// TIA Portal project "Andon L1" (V14)

(* hardware
DEVICE "S7-1200 station_1"  S7-1200 Station
   slot 0: "Rack_0"  S7-1200 Rack  Rack  V1.0
   slot 1: "PLC_1"  CPU 1215C DC/DC/Rly  6ES7 215-1HG40-0XB0  V4.1
*)

// ===== PLC "PLC_1"  CPU 1215C DC/DC/Rly =====

VAR_GLOBAL   // PLC tag table "Default tag table"
   "inverterAssy" AT %I0.0 : Bool;
   "resetTimer" AT %I0.1 : Bool;
   "Tag_3" AT %I0.2 : Bool;
   "System_Byte" AT %MB1 : Byte;
   "FirstScan" AT %M1.0 : Bool;
   "DiagStatusUpdate" AT %M1.1 : Bool;
   "AlwaysTRUE" AT %M1.2 : Bool;
   "AlwaysFALSE" AT %M1.3 : Bool;
   "System_Byte(1)" AT %MB1 : Byte;
   "Clock_Byte" AT %MB0 : Byte;
   "Clock_10Hz" AT %M0.0 : Bool;
   "Clock_5Hz" AT %M0.1 : Bool;
   "Clock_2.5Hz" AT %M0.2 : Bool;
   "Clock_2Hz" AT %M0.3 : Bool;
   "Clock_1.25Hz" AT %M0.4 : Bool;
   "Clock_1Hz" AT %M0.5 : Bool;
   "Clock_0.625Hz" AT %M0.6 : Bool;
   "Clock_0.5Hz" AT %M0.7 : Bool;
   "Send on/off" AT %M10.0 : Bool;
   "Receive enable" AT %M10.1 : Bool;
   "PulseN1" AT %M50.0 : Bool;
   "secStop1" AT %MB20 : Char;
   "PulseN2" AT %M50.1 : Bool;
   "secStop2" AT %MB21 : Char;
   "division1" AT %MB22 : Char;
   "minStop1" AT %MB23 : Char;
   "mResetTimer" AT %M15.0 : Bool;
   "minStop2" AT %MB24 : Char;
   "division2" AT %MB25 : Char;
   "Tag_1" AT %MD20 : DWord;
   "Tag_2" AT %M10.2 : Bool;
   "System_Byte(2)" AT %MB1 : Byte;
   "hourStop2" AT %MB27 : Char;
   "hourStop1" AT %MB26 : Char;
END_VAR

DATA_BLOCK "TCPIP_COMMS_DB"   // DB1
{ S7_Optimized_Access := 'TRUE' }
VERSION : 0.1
// stored: InstanceOfName TCPIP_COMMS
"TCPIP_COMMS"
BEGIN
END_DATA_BLOCK

DATA_BLOCK "DATA"   // DB6
{ S7_Optimized_Access := 'FALSE' }
VERSION : 0.1
   VAR
      Receive : Array[0..1] of Char;
      Send : Array[0..7] of Char;
   END_VAR
BEGIN
END_DATA_BLOCK

// folder: System blocks/Program resources

DATA_BLOCK "PLC_1_Connection_DB"   // DB3
{ S7_Optimized_Access := 'TRUE' }
AUTHOR : SIMATIC
FAMILY : MC7Plus
NAME : TC_IP_v4
VERSION : 1.0
// stored: InstanceOfName TCON_IP_v4
"TCON_IP_v4"
BEGIN
   ID := 1;
   InterfaceId := 64;
   RemotePort := 2000;
   ActiveEstablished := true;
   RemoteAddress.ADDR[1] := 10;
   RemoteAddress.ADDR[2] := 81;
   RemoteAddress.ADDR[3] := 4;
   RemoteAddress.ADDR[4] := 123;
END_DATA_BLOCK

// folder: (top level)

FUNCTION_BLOCK "TCPIP_COMMS"   // FB1, LAD
{ S7_Optimized_Access := 'TRUE' }
VERSION : 0.1
   VAR
      TCON : Struct
         REQ : Bool;
         DONE : Bool;
         BUZY : Bool;
         ERROR : Bool;
         STATUS : UInt;
         DONESAVE : Bool;
      END_STRUCT;
      TDISCON : Struct
         REQ : Bool;
         DONE : Bool;
         BUZY : Bool;
         ERROR : Bool;
         DONESAVE : Bool;
         STATUS : UInt;
      END_STRUCT;
      TSEND : Struct
         REQ : Bool;
         DONE : Bool;
         BUZY : Bool;
         ERROR : Bool;
         DONESAVE : Bool;
         STATUS : UInt;
      END_STRUCT;
      TRCV : Struct
         EN_R : Bool;
         NOR : Bool;
         BUZY : Bool;
         ERROR : Bool;
         STATUS : UInt;
         RCVD_LEN : UDInt;
      END_STRUCT;
      ReceivedString : String;
   END_VAR
   VAR_TEMP
      Temp_1 : Array[0..5] of Char;
   END_VAR
BEGIN

REGION Network 1: TCON
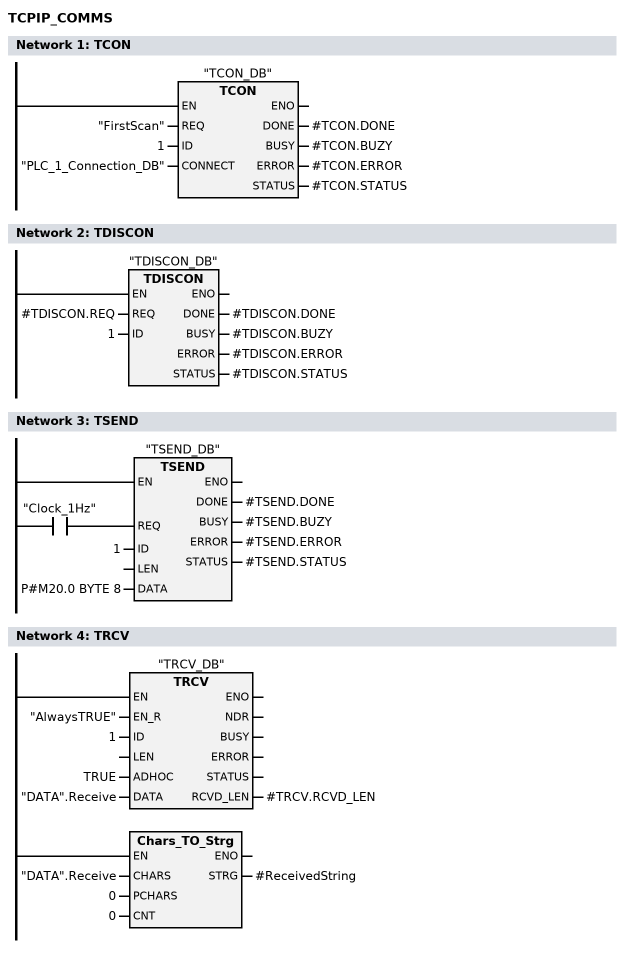
   "TCON_DB"(REQ := "FirstScan",   // TCON
             ID := 1,
             CONNECT := "PLC_1_Connection_DB",
             DONE => #TCON.DONE,
             BUSY => #TCON.BUZY,
             ERROR => #TCON.ERROR,
             STATUS => #TCON.STATUS);
END_REGION

REGION Network 2: TDISCON
   "TDISCON_DB"(REQ := #TDISCON.REQ,   // TDISCON
                ID := 1,
                DONE => #TDISCON.DONE,
                BUSY => #TDISCON.BUZY,
                ERROR => #TDISCON.ERROR,
                STATUS => #TDISCON.STATUS);
END_REGION

REGION Network 3: TSEND
   "TSEND_DB"(REQ := "Clock_1Hz",   // TSEND
              ID := 1,
              DATA := P#M20.0 BYTE 8,
              DONE => #TSEND.DONE,
              BUSY => #TSEND.BUZY,
              ERROR => #TSEND.ERROR,
              STATUS => #TSEND.STATUS);
END_REGION

REGION Network 4: TRCV
   // no SCL statement known for Chars_TO_Strg: written as a call
   "TRCV_DB"(EN_R := "AlwaysTRUE", ID := 1, ADHOC := TRUE, DATA := "DATA".Receive, RCVD_LEN => #TRCV.RCVD_LEN);   // TRCV
   Chars_TO_Strg(Chars := "DATA".Receive, pChars := 0, Cnt := 0, Strg => #ReceivedString);
END_REGION
END_FUNCTION_BLOCK

ORGANIZATION_BLOCK "Main"   // OB1, LAD, ProgramCycle
TITLE = "Main Program Sweep (Cycle)"
{ S7_Optimized_Access := 'TRUE' }
VERSION : 0.1
   VAR_INPUT
      Initial_Call : Bool;   // Initial call of this OB
      Remanence : Bool;   // =True, if remanent data are available
   END_VAR
   VAR_TEMP   // added for the SCL form of the ladder/FBD networks
      _w1 : Bool;
      _w2 : Bool;
      _w3 : Bool;
      _w4 : Bool;
      _w5 : Bool;
      _w6 : Bool;
      _w7 : Bool;
   END_VAR
BEGIN

REGION Network 1
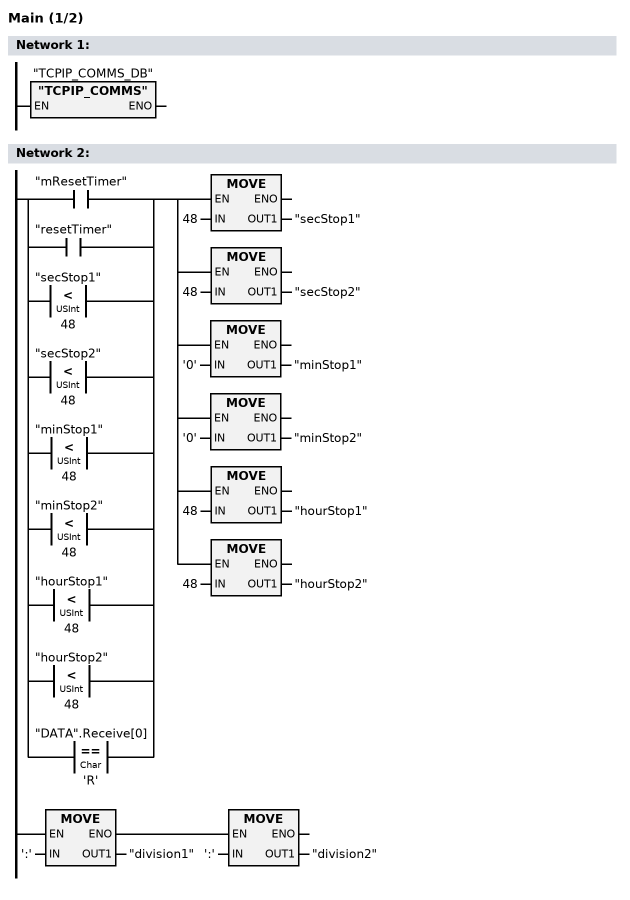
   RUNG wire#powerrail
      "TCPIP_COMMS_DB"()
   END_RUNG
   // the same network as SCL:
   "TCPIP_COMMS_DB"();   // "TCPIP_COMMS"
END_REGION

REGION Network 2
   RUNG wire#powerrail
      Contact( "mResetTimer" )
      wire#w1
      Move(in := 48, out1 => "secStop1")
   END_RUNG
   RUNG wire#powerrail
      Contact( "resetTimer" )
   END_RUNG wire#w1
   RUNG wire#powerrail
      { S7_Templates := "SrcType := USInt" } LT_Contact(in1 := "secStop1", in2 := 48)
   END_RUNG wire#w1
   RUNG wire#powerrail
      { S7_Templates := "SrcType := USInt" } LT_Contact(in1 := "secStop2", in2 := 48)
   END_RUNG wire#w1
   RUNG wire#powerrail
      { S7_Templates := "SrcType := USInt" } LT_Contact(in1 := "minStop1", in2 := 48)
   END_RUNG wire#w1
   RUNG wire#powerrail
      { S7_Templates := "SrcType := USInt" } LT_Contact(in1 := "minStop2", in2 := 48)
   END_RUNG wire#w1
   RUNG wire#powerrail
      { S7_Templates := "SrcType := USInt" } LT_Contact(in1 := "hourStop1", in2 := 48)
   END_RUNG wire#w1
   RUNG wire#powerrail
      { S7_Templates := "SrcType := USInt" } LT_Contact(in1 := "hourStop2", in2 := 48)
   END_RUNG wire#w1
   RUNG wire#powerrail
      { S7_Templates := "SrcType := Char" } EQ_Contact(in1 := "DATA".Receive[0], in2 := 'R')
   END_RUNG wire#w1
   RUNG wire#w1
      Move(in := 48, out1 => "secStop2")
   END_RUNG
   RUNG wire#w1
      Move(in := '0', out1 => "minStop1")
   END_RUNG
   RUNG wire#w1
      Move(in := '0', out1 => "minStop2")
   END_RUNG
   RUNG wire#w1
      Move(in := 48, out1 => "hourStop1")
   END_RUNG
   RUNG wire#w1
      Move(in := 48, out1 => "hourStop2")
   END_RUNG
   RUNG wire#powerrail
      Move(in := ':', out1 => "division1")
      Move(in := ':', out1 => "division2")
   END_RUNG
   // the same network as SCL:
   #_w1 := "mResetTimer" OR "resetTimer" OR ("secStop1" < 48) OR ("secStop2" < 48) OR ("minStop1" < 48) OR ("minStop2" < 48) OR ("hourStop1" < 48) OR ("hourStop2" < 48) OR ("DATA".Receive[0] = 'R');
   IF #_w1 THEN
       "secStop1" := 48;
       "secStop2" := 48;
       "minStop1" := '0';
       "minStop2" := '0';
       "hourStop1" := 48;
       "hourStop2" := 48;
   END_IF;
   "division1" := ':';
   "division2" := ':';
END_REGION

REGION Network 3: Seconds
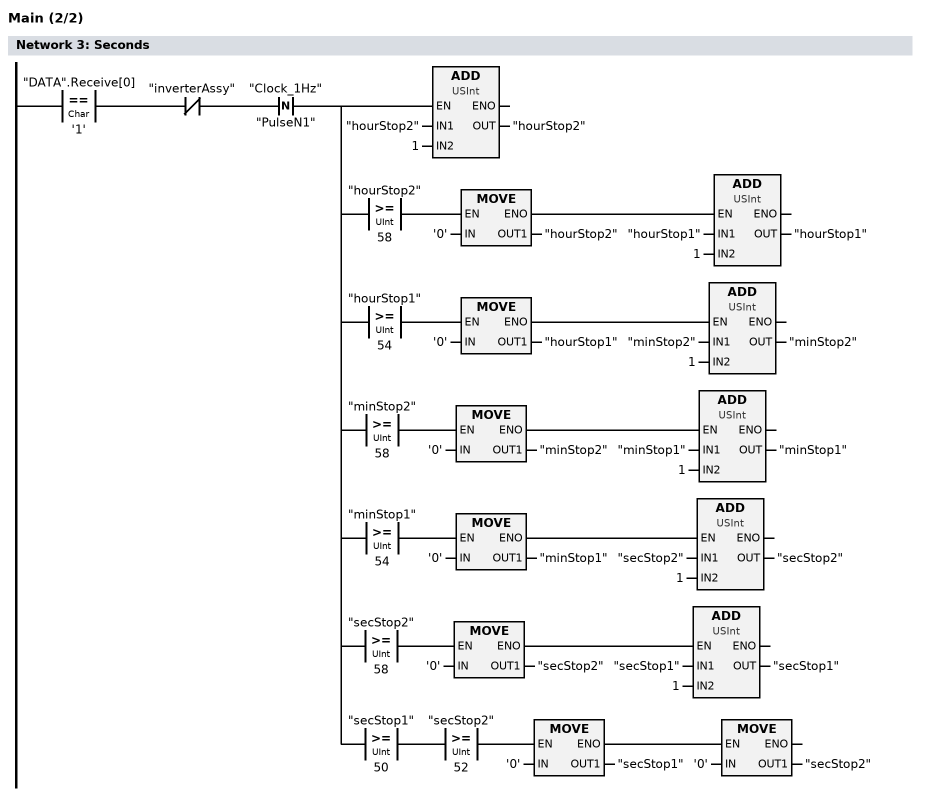
   RUNG wire#powerrail
      { S7_Templates := "SrcType := Char" } EQ_Contact(in1 := "DATA".Receive[0], in2 := '1')
      I_Contact( "inverterAssy" )
      N_Contact(operand := "Clock_1Hz", bit := "PulseN1")
      wire#w1
      { S7_Templates := "SrcType := USInt" } Add(in1 := "hourStop2", in2 := 1, out => "hourStop2")
   END_RUNG
   RUNG wire#w1
      { S7_Templates := "SrcType := UInt" } GE_Contact(in1 := "hourStop2", in2 := 58)
      Move(in := '0', out1 => "hourStop2")
      { S7_Templates := "SrcType := USInt" } Add(in1 := "hourStop1", in2 := 1, out => "hourStop1")
   END_RUNG
   RUNG wire#w1
      { S7_Templates := "SrcType := UInt" } GE_Contact(in1 := "hourStop1", in2 := 54)
      Move(in := '0', out1 => "hourStop1")
      { S7_Templates := "SrcType := USInt" } Add(in1 := "minStop2", in2 := 1, out => "minStop2")
   END_RUNG
   RUNG wire#w1
      { S7_Templates := "SrcType := UInt" } GE_Contact(in1 := "minStop2", in2 := 58)
      Move(in := '0', out1 => "minStop2")
      { S7_Templates := "SrcType := USInt" } Add(in1 := "minStop1", in2 := 1, out => "minStop1")
   END_RUNG
   RUNG wire#w1
      { S7_Templates := "SrcType := UInt" } GE_Contact(in1 := "minStop1", in2 := 54)
      Move(in := '0', out1 => "minStop1")
      { S7_Templates := "SrcType := USInt" } Add(in1 := "secStop2", in2 := 1, out => "secStop2")
   END_RUNG
   RUNG wire#w1
      { S7_Templates := "SrcType := UInt" } GE_Contact(in1 := "secStop2", in2 := 58)
      Move(in := '0', out1 => "secStop2")
      { S7_Templates := "SrcType := USInt" } Add(in1 := "secStop1", in2 := 1, out => "secStop1")
   END_RUNG
   RUNG wire#w1
      { S7_Templates := "SrcType := UInt" } GE_Contact(in1 := "secStop1", in2 := 50)
      { S7_Templates := "SrcType := UInt" } GE_Contact(in1 := "secStop2", in2 := 52)
      Move(in := '0', out1 => "secStop1")
      Move(in := '0', out1 => "secStop2")
   END_RUNG
   // the same network as SCL:
   #_w1 := ("DATA".Receive[0] = '1') AND NOT "inverterAssy" AND NOT "Clock_1Hz" AND "PulseN1";   // falling edge of "Clock_1Hz"
   "PulseN1" := "Clock_1Hz";
   IF #_w1 THEN "hourStop2" := "hourStop2" + 1; END_IF;
   #_w2 := #_w1 AND ("hourStop2" >= 58);
   IF #_w2 THEN
       "hourStop2" := '0';
       "hourStop1" := "hourStop1" + 1;
   END_IF;
   #_w3 := #_w1 AND ("hourStop1" >= 54);
   IF #_w3 THEN
       "hourStop1" := '0';
       "minStop2" := "minStop2" + 1;
   END_IF;
   #_w4 := #_w1 AND ("minStop2" >= 58);
   IF #_w4 THEN
       "minStop2" := '0';
       "minStop1" := "minStop1" + 1;
   END_IF;
   #_w5 := #_w1 AND ("minStop1" >= 54);
   IF #_w5 THEN
       "minStop1" := '0';
       "secStop2" := "secStop2" + 1;
   END_IF;
   #_w6 := #_w1 AND ("secStop2" >= 58);
   IF #_w6 THEN
       "secStop2" := '0';
       "secStop1" := "secStop1" + 1;
   END_IF;
   #_w7 := #_w1 AND ("secStop1" >= 50) AND ("secStop2" >= 52);
   IF #_w7 THEN
       "secStop1" := '0';
       "secStop2" := '0';
   END_IF;
END_REGION

REGION Network 4: Hour
END_REGION
END_ORGANIZATION_BLOCK